Fanuc KAREL source: kt00411.KL

-- PROVISIONAL review KL for V770-1; original PC SHA256 e1cef26231a4f35d7fcf0aa5f754eef85f7f66adad45673cb18baf1ad62d32b8
-- Incomplete behavior may be omitted. Consult companion uncertainty JSON. Do not deploy.
PROGRAM KT00411
%NOLOCKGROUP
VAR
  I2 : INTEGER
  OUT : BOOLEAN
-- UNRESOLVED_DECL Y1 type=002018
BEGIN
  -- UNRESOLVED_PC offsets 5-19; opcodes 2E,22,9D,33,B2
  -- UNRESOLVED_PC offsets 24-35; opcodes 2E,23
  -- UNRESOLVED_PC offsets 40-62; opcodes 22,9D,33,B1,21,5B,23
  -- UNRESOLVED_PC offsets 67-71; opcodes 7F
END KT00411
